PROGRAM Energieverbrauch
VAR
	EnergieverbrauchMotor1: REAL;
	EnergieverbrauchMotor2: REAL;
	EnergieverbrauchMotor3: REAL;
	EnergieverbrauchEbus:	REAL;
	
	LeistungMotor1: INT;
	LeistungMotor2: INT;
	LeistungMotor3: INT;
	LeistungEbus:	INT;
END_VAR

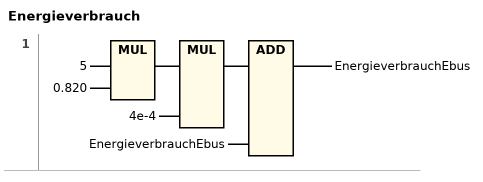
// NETWORK 1
EnergieverbrauchEbus := (5 * 0.820) * (4e-4) + EnergieverbrauchEbus;

END_PROGRAM

(* stored: Version 1.1.0.1, ProductVersion 3.1.4022.3
   POU Energieverbrauch: Id {409b7099-9e0c-49d7-87be-a50544e33f1e}, SpecialFunc None *)
